(* Logix 5000 project; controller R5_CSS vendor 1 type 14 code 74 rev 19.11; software revision 19.01; part 17 of 20 *)
(* tags used below, declared in another part *)
   AlarmMaster : DINT;
   AllowHeatersWhenEmpty : BOOL;
   GTL_TDAHH_MinSP : REAL;
   HT_FAULT : BOOL;
   LC302 : LEVEL_CONTROL;   // COALESCER OIL CHAMBER LEVEL CONTROL
   MV301 : ValveControl_TwoWay;
   P302A : PUMP_CONTROL;
   P302B : PUMP_CONTROL;
   PID_JHE319 : PID;   // TEMPERATURE CONTROL OUPUT FOR JHE313B PID
   PID_JHE319_TON : TIMER;
   PID_TC215_TON : TIMER;
   PRU_TT404 : REAL[10];
   PRUA_READ : INT[30];
   TC112A : TEMP_CONTROL;
   TC121 : TEMP_CONTROL;
   TC121A : TEMP_CONTROL;   // GTL FROM PRUA TEMPERATURE CONTROL
   TC135 : TEMP_CONTROL;
   TC136 : TEMP_CONTROL;
   TC137 : TEMP_CONTROL;
   TC215 : TEMP_CONTROL;   // OVERHEAD CONDENSER CHILLED WATER TEMPERATURE TRANSMITTER CONTROL
   TC215_AUTO_ONS1 : BOOL;
   TC215_MANUAL_ONS1 : BOOL;
   TC313A : TEMP_CONTROL;   // PRIMARY COALESCER SEPARATOR TEMPERATURE CONTROL
   TC319 : TEMP_CONTROL;   // COALESCER OIL CHAMBER PROCESS TEMPERATURE CONTROL
   TC319_AUTO_Ons : BOOL;
   TC319_AUTO_Ons1 : BOOL;
   TC319_HeaterDisabled : BOOL;
   TC319_MANUAL_Ons : BOOL;
   TC319_START_TON : TIMER;
   TC319A : TEMP_CONTROL;   // COALESCER OIL CHAMBER SHEATH TEMPERATURE
   TCV215_PID : PID;
   TMR_FAULT : DINT;
(* MainProgram, continued *)

ROUTINE TC112A_CoalWaterHeaterBundleTemp   (* ladder *)
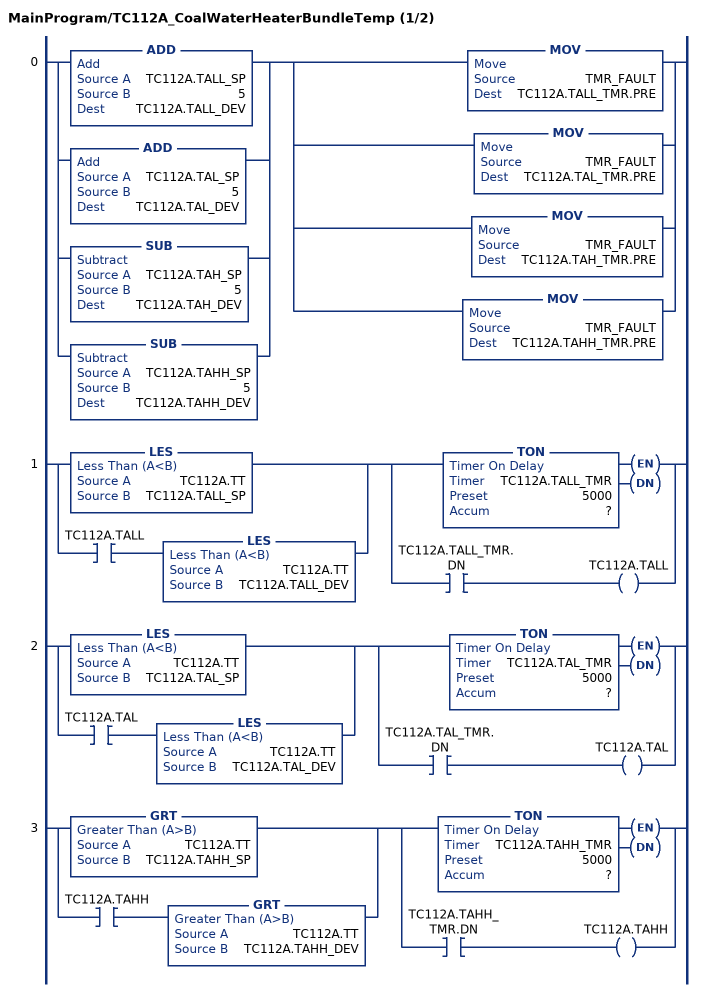
   0: [ADD(TC112A.TALL_SP,5,TC112A.TALL_DEV) ,ADD(TC112A.TAL_SP,5,TC112A.TAL_DEV) ,SUB(TC112A.TAH_SP,5,TC112A.TAH_DEV) ,SUB(TC112A.TAHH_SP,5,TC112A.TAHH_DEV) ][MOV(TMR_FAULT,TC112A.TALL_TMR.PRE) ,MOV(TMR_FAULT,TC112A.TAL_TMR.PRE) ,MOV(TMR_FAULT,TC112A.TAH_TMR.PRE) ,MOV(TMR_FAULT,TC112A.TAHH_TMR.PRE) ];
   1: [LES(TC112A.TT,TC112A.TALL_SP) ,XIC(TC112A.TALL) LES(TC112A.TT,TC112A.TALL_DEV) ][TON(TC112A.TALL_TMR,?,?) ,XIC(TC112A.TALL_TMR.DN) OTE(TC112A.TALL) ];
   2: [LES(TC112A.TT,TC112A.TAL_SP) ,XIC(TC112A.TAL) LES(TC112A.TT,TC112A.TAL_DEV) ][TON(TC112A.TAL_TMR,?,?) ,XIC(TC112A.TAL_TMR.DN) OTE(TC112A.TAL) ];
   3: [GRT(TC112A.TT,TC112A.TAHH_SP) ,XIC(TC112A.TAHH) GRT(TC112A.TT,TC112A.TAHH_DEV) ][TON(TC112A.TAHH_TMR,?,?) ,XIC(TC112A.TAHH_TMR.DN) OTE(TC112A.TAHH) ];
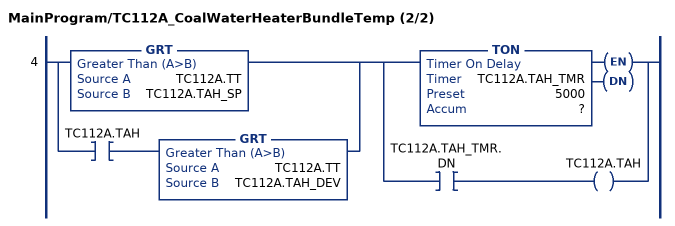
   4: [GRT(TC112A.TT,TC112A.TAH_SP) ,XIC(TC112A.TAH) GRT(TC112A.TT,TC112A.TAH_DEV) ][TON(TC112A.TAH_TMR,?,?) ,XIC(TC112A.TAH_TMR.DN) OTE(TC112A.TAH) ];
END_ROUTINE

ROUTINE TC135_GTL1_Temperature   (* ladder *)
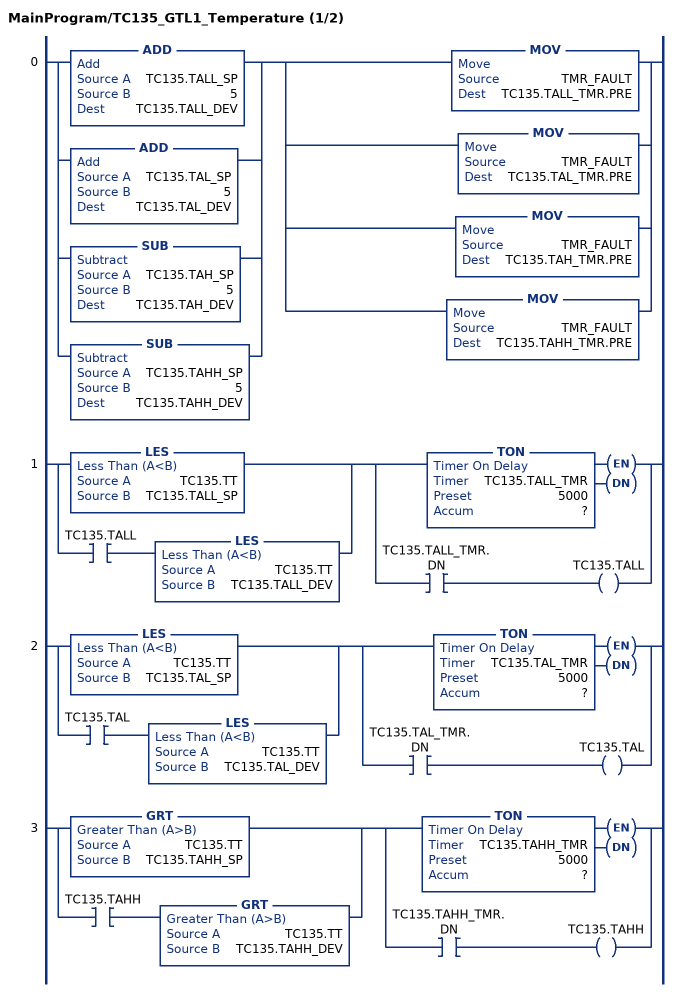
   0: [ADD(TC135.TALL_SP,5,TC135.TALL_DEV) ,ADD(TC135.TAL_SP,5,TC135.TAL_DEV) ,SUB(TC135.TAH_SP,5,TC135.TAH_DEV) ,SUB(TC135.TAHH_SP,5,TC135.TAHH_DEV) ][MOV(TMR_FAULT,TC135.TALL_TMR.PRE) ,MOV(TMR_FAULT,TC135.TAL_TMR.PRE) ,MOV(TMR_FAULT,TC135.TAH_TMR.PRE) ,MOV(TMR_FAULT,TC135.TAHH_TMR.PRE) ];
   1: [LES(TC135.TT,TC135.TALL_SP) ,XIC(TC135.TALL) LES(TC135.TT,TC135.TALL_DEV) ][TON(TC135.TALL_TMR,?,?) ,XIC(TC135.TALL_TMR.DN) OTE(TC135.TALL) ];
   2: [LES(TC135.TT,TC135.TAL_SP) ,XIC(TC135.TAL) LES(TC135.TT,TC135.TAL_DEV) ][TON(TC135.TAL_TMR,?,?) ,XIC(TC135.TAL_TMR.DN) OTE(TC135.TAL) ];
   3: [GRT(TC135.TT,TC135.TAHH_SP) ,XIC(TC135.TAHH) GRT(TC135.TT,TC135.TAHH_DEV) ][TON(TC135.TAHH_TMR,?,?) ,XIC(TC135.TAHH_TMR.DN) OTE(TC135.TAHH) ];
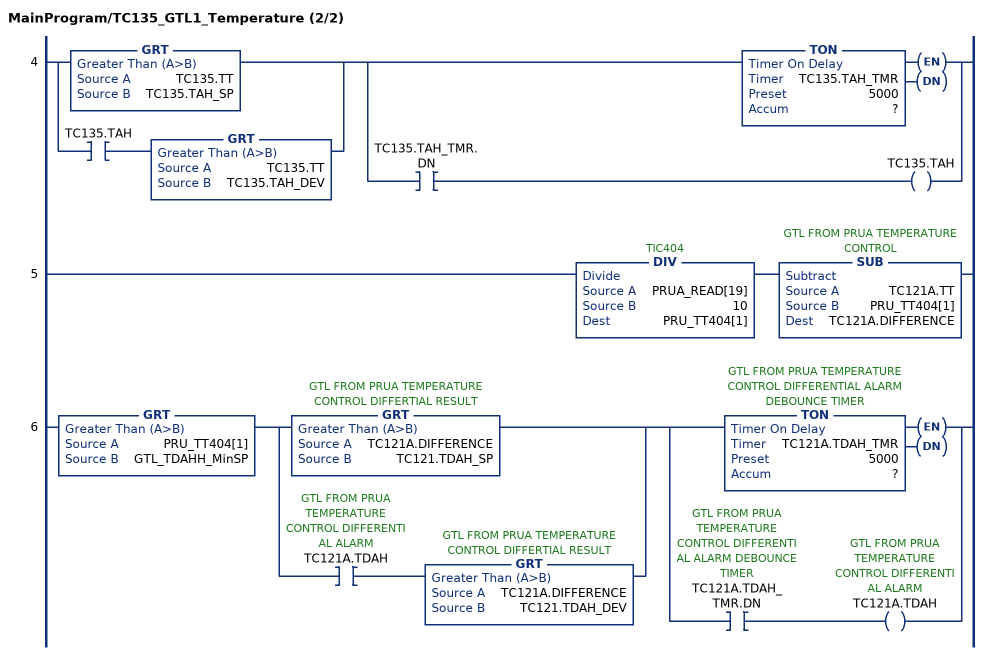
   4: [GRT(TC135.TT,TC135.TAH_SP) ,XIC(TC135.TAH) GRT(TC135.TT,TC135.TAH_DEV) ][TON(TC135.TAH_TMR,?,?) ,XIC(TC135.TAH_TMR.DN) OTE(TC135.TAH) ];
   5: DIV(PRUA_READ[19],10,PRU_TT404[1])SUB(TC121A.TT,PRU_TT404[1],TC121A.DIFFERENCE);
   6: GRT(PRU_TT404[1],GTL_TDAHH_MinSP)[GRT(TC121A.DIFFERENCE,TC121.TDAH_SP) ,XIC(TC121A.TDAH) GRT(TC121A.DIFFERENCE,TC121.TDAH_DEV) ][TON(TC121A.TDAH_TMR,?,?) ,XIC(TC121A.TDAH_TMR.DN) OTE(TC121A.TDAH) ];
END_ROUTINE

ROUTINE TC136_GTL2_Temperature   (* ladder *)
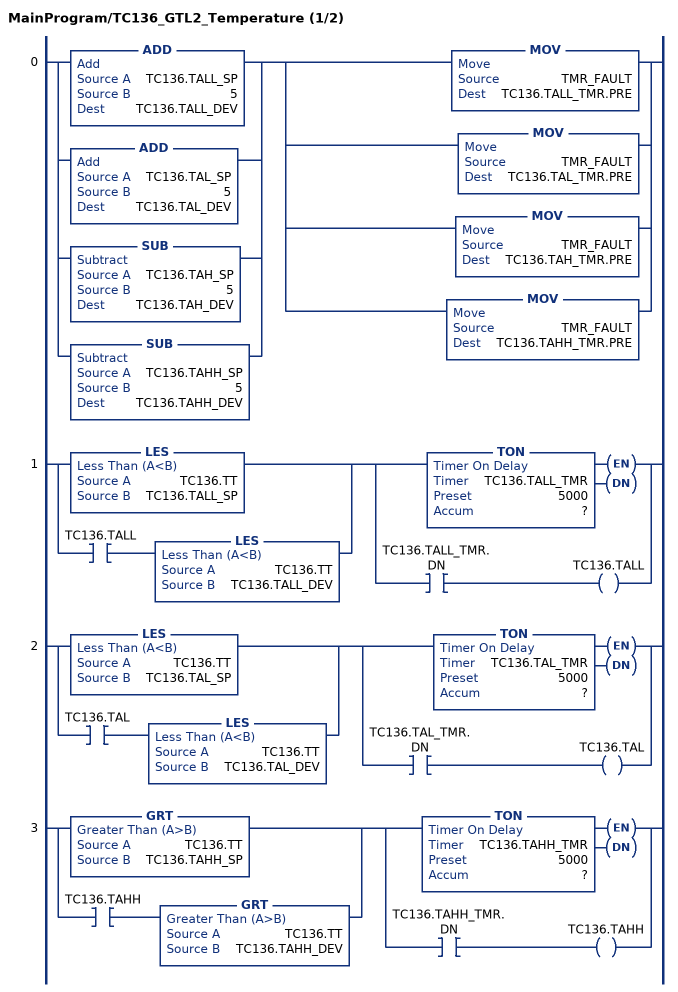
   0: [ADD(TC136.TALL_SP,5,TC136.TALL_DEV) ,ADD(TC136.TAL_SP,5,TC136.TAL_DEV) ,SUB(TC136.TAH_SP,5,TC136.TAH_DEV) ,SUB(TC136.TAHH_SP,5,TC136.TAHH_DEV) ][MOV(TMR_FAULT,TC136.TALL_TMR.PRE) ,MOV(TMR_FAULT,TC136.TAL_TMR.PRE) ,MOV(TMR_FAULT,TC136.TAH_TMR.PRE) ,MOV(TMR_FAULT,TC136.TAHH_TMR.PRE) ];
   1: [LES(TC136.TT,TC136.TALL_SP) ,XIC(TC136.TALL) LES(TC136.TT,TC136.TALL_DEV) ][TON(TC136.TALL_TMR,?,?) ,XIC(TC136.TALL_TMR.DN) OTE(TC136.TALL) ];
   2: [LES(TC136.TT,TC136.TAL_SP) ,XIC(TC136.TAL) LES(TC136.TT,TC136.TAL_DEV) ][TON(TC136.TAL_TMR,?,?) ,XIC(TC136.TAL_TMR.DN) OTE(TC136.TAL) ];
   3: [GRT(TC136.TT,TC136.TAHH_SP) ,XIC(TC136.TAHH) GRT(TC136.TT,TC136.TAHH_DEV) ][TON(TC136.TAHH_TMR,?,?) ,XIC(TC136.TAHH_TMR.DN) OTE(TC136.TAHH) ];
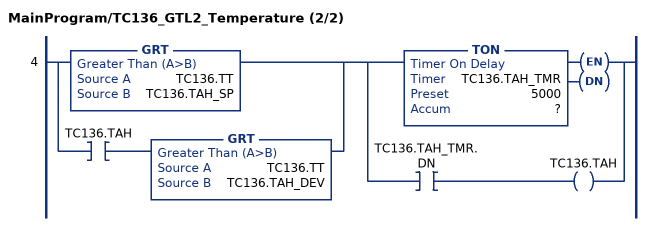
   4: [GRT(TC136.TT,TC136.TAH_SP) ,XIC(TC136.TAH) GRT(TC136.TT,TC136.TAH_DEV) ][TON(TC136.TAH_TMR,?,?) ,XIC(TC136.TAH_TMR.DN) OTE(TC136.TAH) ];
END_ROUTINE

ROUTINE TC137_GTL3_Temperature   (* ladder *)
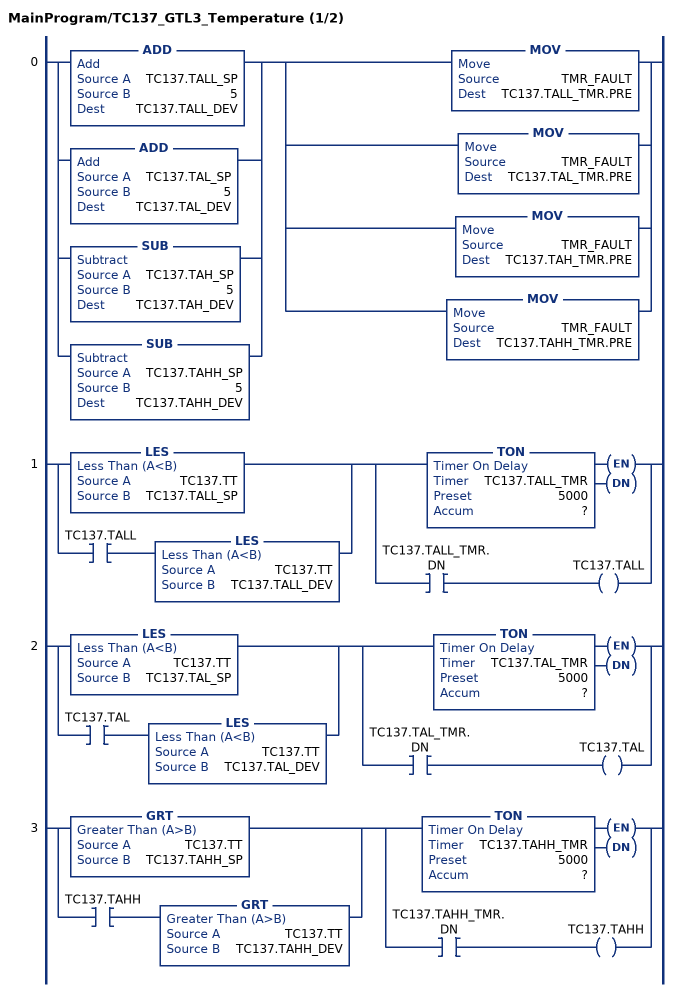
   0: [ADD(TC137.TALL_SP,5,TC137.TALL_DEV) ,ADD(TC137.TAL_SP,5,TC137.TAL_DEV) ,SUB(TC137.TAH_SP,5,TC137.TAH_DEV) ,SUB(TC137.TAHH_SP,5,TC137.TAHH_DEV) ][MOV(TMR_FAULT,TC137.TALL_TMR.PRE) ,MOV(TMR_FAULT,TC137.TAL_TMR.PRE) ,MOV(TMR_FAULT,TC137.TAH_TMR.PRE) ,MOV(TMR_FAULT,TC137.TAHH_TMR.PRE) ];
   1: [LES(TC137.TT,TC137.TALL_SP) ,XIC(TC137.TALL) LES(TC137.TT,TC137.TALL_DEV) ][TON(TC137.TALL_TMR,?,?) ,XIC(TC137.TALL_TMR.DN) OTE(TC137.TALL) ];
   2: [LES(TC137.TT,TC137.TAL_SP) ,XIC(TC137.TAL) LES(TC137.TT,TC137.TAL_DEV) ][TON(TC137.TAL_TMR,?,?) ,XIC(TC137.TAL_TMR.DN) OTE(TC137.TAL) ];
   3: [GRT(TC137.TT,TC137.TAHH_SP) ,XIC(TC137.TAHH) GRT(TC137.TT,TC137.TAHH_DEV) ][TON(TC137.TAHH_TMR,?,?) ,XIC(TC137.TAHH_TMR.DN) OTE(TC137.TAHH) ];
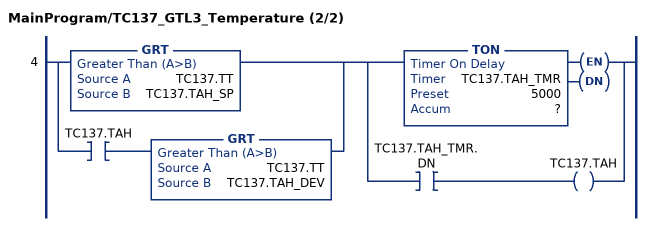
   4: [GRT(TC137.TT,TC137.TAH_SP) ,XIC(TC137.TAH) GRT(TC137.TT,TC137.TAH_DEV) ][TON(TC137.TAH_TMR,?,?) ,XIC(TC137.TAH_TMR.DN) OTE(TC137.TAH) ];
END_ROUTINE

ROUTINE TC215_OverheadCondTemp_PID   (* ladder *)
// NonCondensable Process Gas Temperature Control
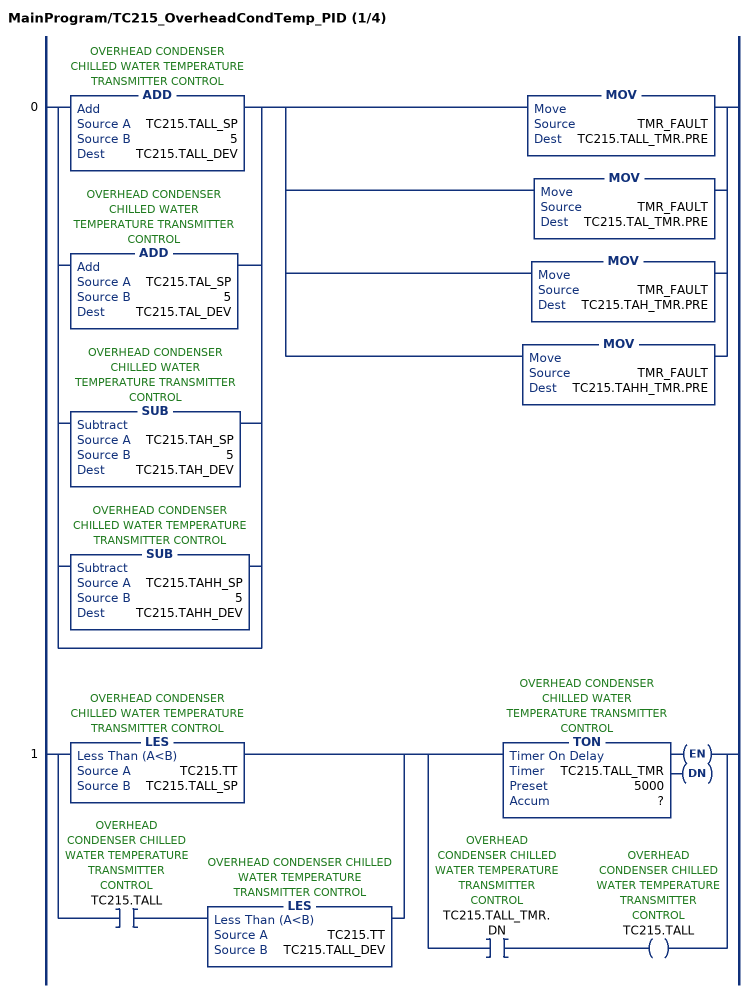
   0: [ADD(TC215.TALL_SP,5,TC215.TALL_DEV) ,ADD(TC215.TAL_SP,5,TC215.TAL_DEV) ,SUB(TC215.TAH_SP,5,TC215.TAH_DEV) ,SUB(TC215.TAHH_SP,5,TC215.TAHH_DEV) ,][MOV(TMR_FAULT,TC215.TALL_TMR.PRE) ,MOV(TMR_FAULT,TC215.TAL_TMR.PRE) ,MOV(TMR_FAULT,TC215.TAH_TMR.PRE) ,MOV(TMR_FAULT,TC215.TAHH_TMR.PRE) ];
   1: [LES(TC215.TT,TC215.TALL_SP) ,XIC(TC215.TALL) LES(TC215.TT,TC215.TALL_DEV) ][TON(TC215.TALL_TMR,?,?) ,XIC(TC215.TALL_TMR.DN) OTE(TC215.TALL) ];
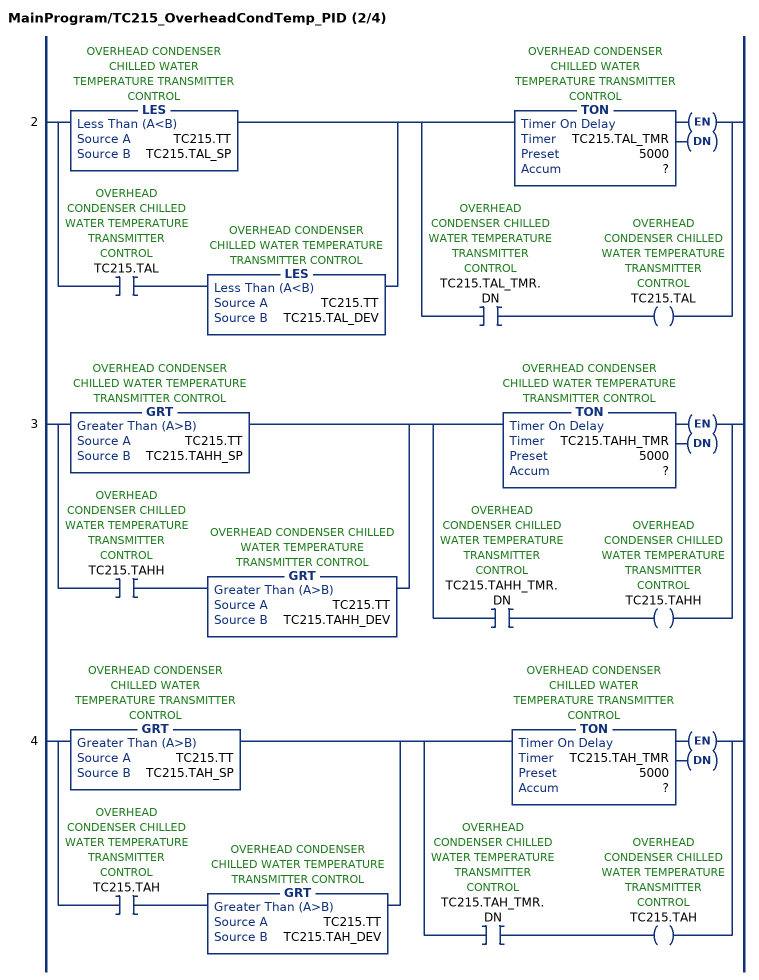
   2: [LES(TC215.TT,TC215.TAL_SP) ,XIC(TC215.TAL) LES(TC215.TT,TC215.TAL_DEV) ][TON(TC215.TAL_TMR,?,?) ,XIC(TC215.TAL_TMR.DN) OTE(TC215.TAL) ];
   3: [GRT(TC215.TT,TC215.TAHH_SP) ,XIC(TC215.TAHH) GRT(TC215.TT,TC215.TAHH_DEV) ][TON(TC215.TAHH_TMR,?,?) ,XIC(TC215.TAHH_TMR.DN) OTE(TC215.TAHH) ];
   4: [GRT(TC215.TT,TC215.TAH_SP) ,XIC(TC215.TAH) GRT(TC215.TT,TC215.TAH_DEV) ][TON(TC215.TAH_TMR,?,?) ,XIC(TC215.TAH_TMR.DN) OTE(TC215.TAH) ];
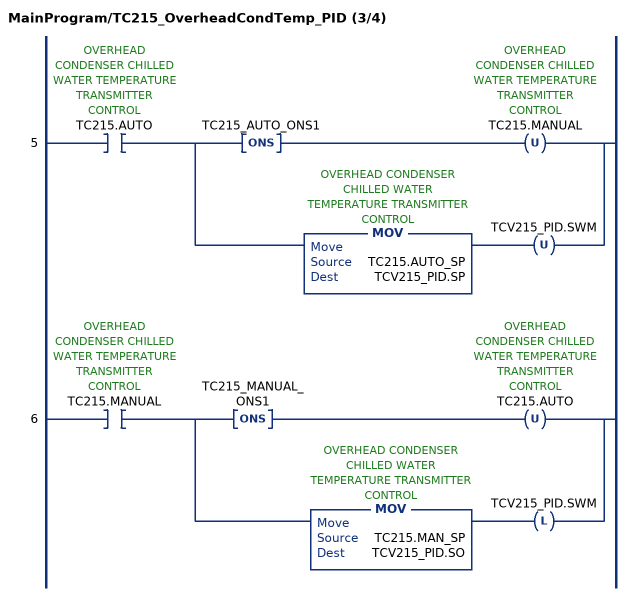
   5: XIC(TC215.AUTO)[ONS(TC215_AUTO_ONS1) OTU(TC215.MANUAL) ,MOV(TC215.AUTO_SP,TCV215_PID.SP) OTU(TCV215_PID.SWM) ];
   6: XIC(TC215.MANUAL)[ONS(TC215_MANUAL_ONS1) OTU(TC215.AUTO) ,MOV(TC215.MAN_SP,TCV215_PID.SO) OTL(TCV215_PID.SWM) ];
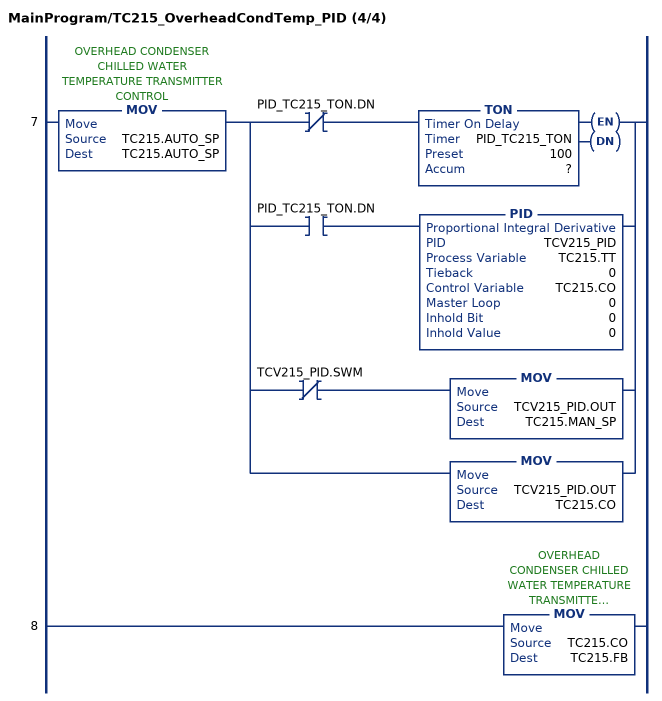
   7: MOV(TC215.AUTO_SP,TC215.AUTO_SP)[XIO(PID_TC215_TON.DN) TON(PID_TC215_TON,?,?) ,XIC(PID_TC215_TON.DN) PID(TCV215_PID,TC215.TT,0,TC215.CO,0,0,0) ,XIO(TCV215_PID.SWM) MOV(TCV215_PID.OUT,TC215.MAN_SP) ,MOV(TCV215_PID.OUT,TC215.CO) ];
   8: MOV(TC215.CO,TC215.FB);
END_ROUTINE

ROUTINE TC313A_CoalPriChamberTemperature   (* ladder *)
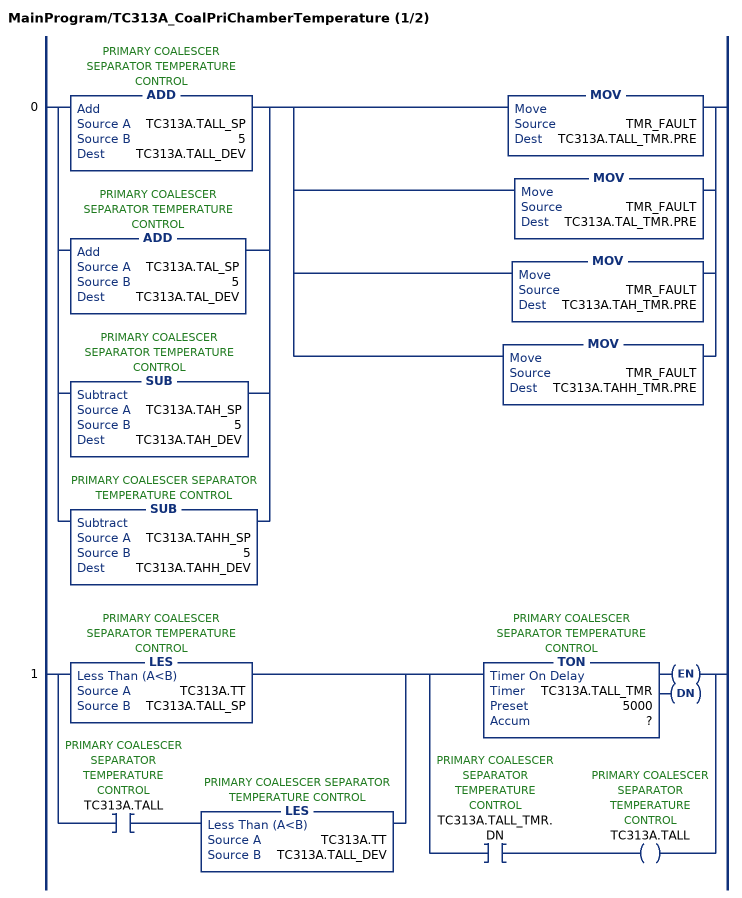
   0: [ADD(TC313A.TALL_SP,5,TC313A.TALL_DEV) ,ADD(TC313A.TAL_SP,5,TC313A.TAL_DEV) ,SUB(TC313A.TAH_SP,5,TC313A.TAH_DEV) ,SUB(TC313A.TAHH_SP,5,TC313A.TAHH_DEV) ][MOV(TMR_FAULT,TC313A.TALL_TMR.PRE) ,MOV(TMR_FAULT,TC313A.TAL_TMR.PRE) ,MOV(TMR_FAULT,TC313A.TAH_TMR.PRE) ,MOV(TMR_FAULT,TC313A.TAHH_TMR.PRE) ];
   1: [LES(TC313A.TT,TC313A.TALL_SP) ,XIC(TC313A.TALL) LES(TC313A.TT,TC313A.TALL_DEV) ][TON(TC313A.TALL_TMR,?,?) ,XIC(TC313A.TALL_TMR.DN) OTE(TC313A.TALL) ];
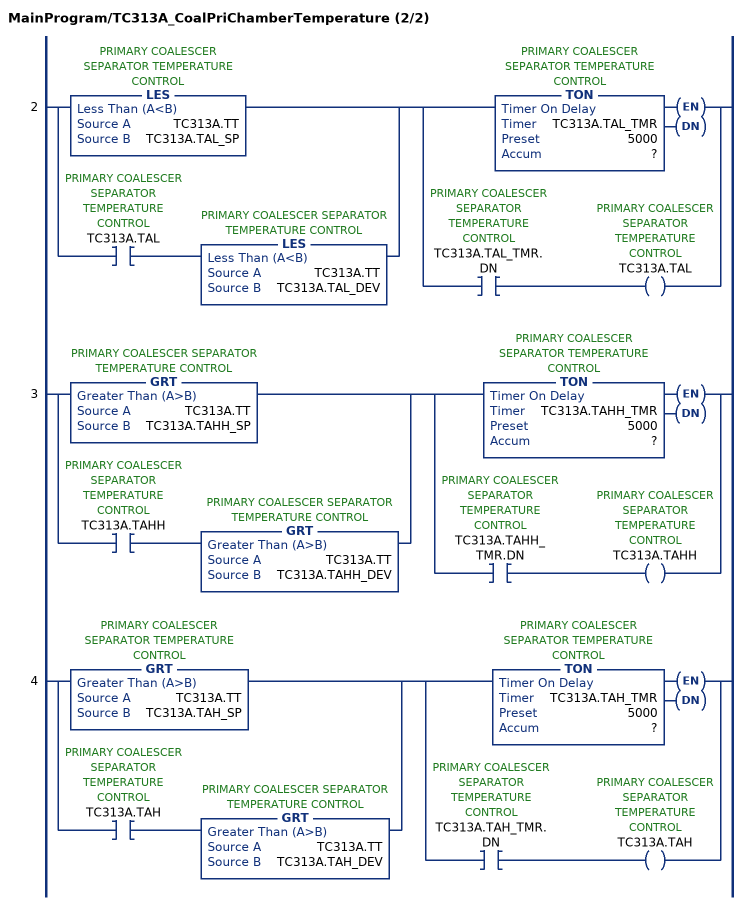
   2: [LES(TC313A.TT,TC313A.TAL_SP) ,XIC(TC313A.TAL) LES(TC313A.TT,TC313A.TAL_DEV) ][TON(TC313A.TAL_TMR,?,?) ,XIC(TC313A.TAL_TMR.DN) OTE(TC313A.TAL) ];
   3: [GRT(TC313A.TT,TC313A.TAHH_SP) ,XIC(TC313A.TAHH) GRT(TC313A.TT,TC313A.TAHH_DEV) ][TON(TC313A.TAHH_TMR,?,?) ,XIC(TC313A.TAHH_TMR.DN) OTE(TC313A.TAHH) ];
   4: [GRT(TC313A.TT,TC313A.TAH_SP) ,XIC(TC313A.TAH) GRT(TC313A.TT,TC313A.TAH_DEV) ][TON(TC313A.TAH_TMR,?,?) ,XIC(TC313A.TAH_TMR.DN) OTE(TC313A.TAH) ];
END_ROUTINE

ROUTINE TC319_OilProductTemperature_PID   (* ladder *)
// OIL TRANSFER CHAMBER HEAT CONTROL
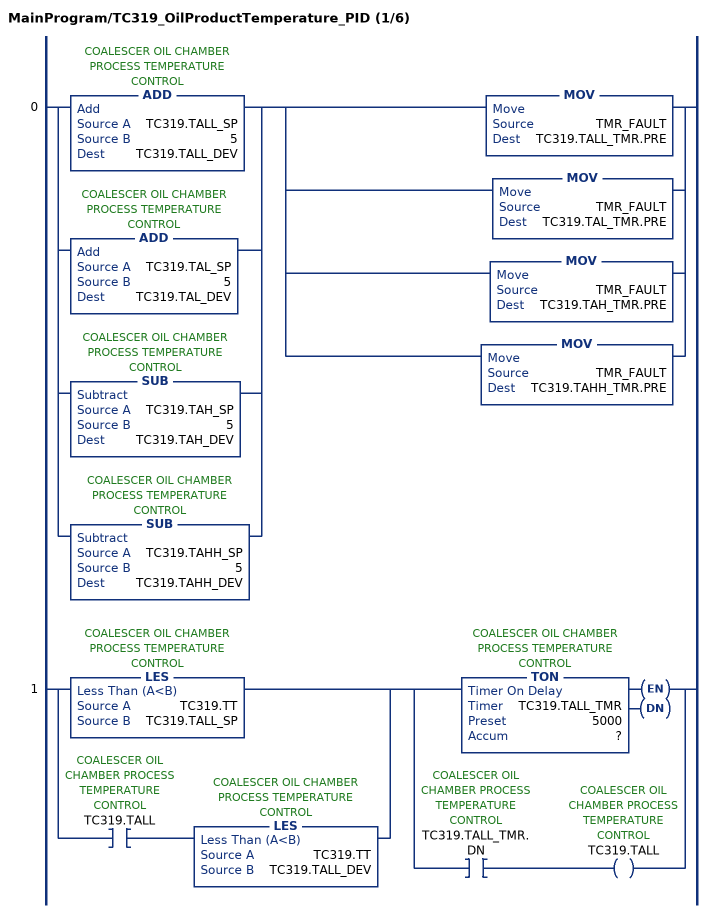
   0: [ADD(TC319.TALL_SP,5,TC319.TALL_DEV) ,ADD(TC319.TAL_SP,5,TC319.TAL_DEV) ,SUB(TC319.TAH_SP,5,TC319.TAH_DEV) ,SUB(TC319.TAHH_SP,5,TC319.TAHH_DEV) ][MOV(TMR_FAULT,TC319.TALL_TMR.PRE) ,MOV(TMR_FAULT,TC319.TAL_TMR.PRE) ,MOV(TMR_FAULT,TC319.TAH_TMR.PRE) ,MOV(TMR_FAULT,TC319.TAHH_TMR.PRE) ];
   1: [LES(TC319.TT,TC319.TALL_SP) ,XIC(TC319.TALL) LES(TC319.TT,TC319.TALL_DEV) ][TON(TC319.TALL_TMR,?,?) ,XIC(TC319.TALL_TMR.DN) OTE(TC319.TALL) ];
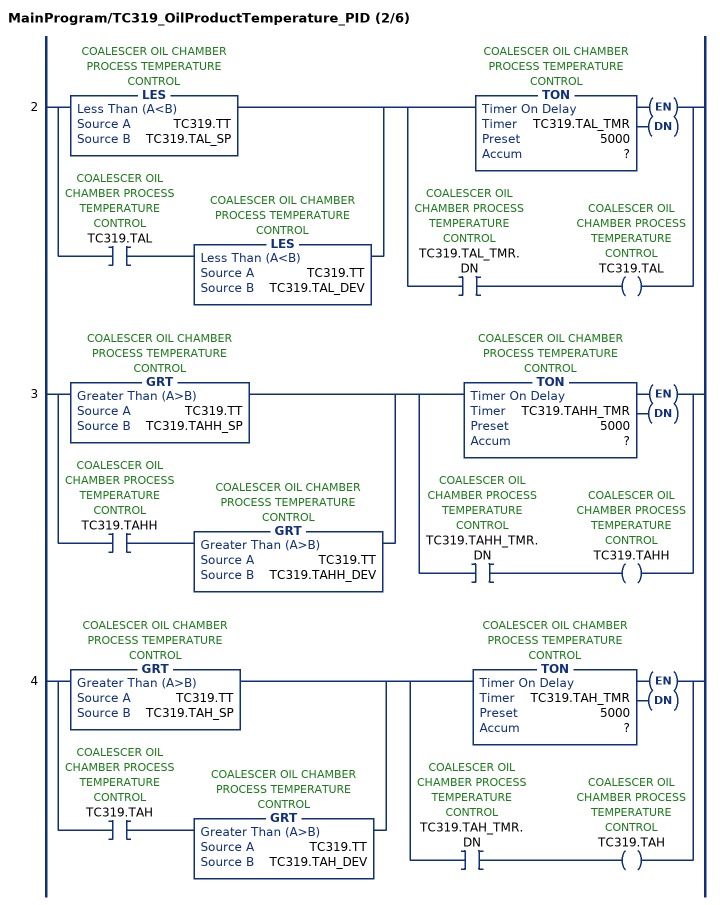
   2: [LES(TC319.TT,TC319.TAL_SP) ,XIC(TC319.TAL) LES(TC319.TT,TC319.TAL_DEV) ][TON(TC319.TAL_TMR,?,?) ,XIC(TC319.TAL_TMR.DN) OTE(TC319.TAL) ];
   3: [GRT(TC319.TT,TC319.TAHH_SP) ,XIC(TC319.TAHH) GRT(TC319.TT,TC319.TAHH_DEV) ][TON(TC319.TAHH_TMR,?,?) ,XIC(TC319.TAHH_TMR.DN) OTE(TC319.TAHH) ];
   4: [GRT(TC319.TT,TC319.TAH_SP) ,XIC(TC319.TAH) GRT(TC319.TT,TC319.TAH_DEV) ][TON(TC319.TAH_TMR,?,?) ,XIC(TC319.TAH_TMR.DN) OTE(TC319.TAH) ];
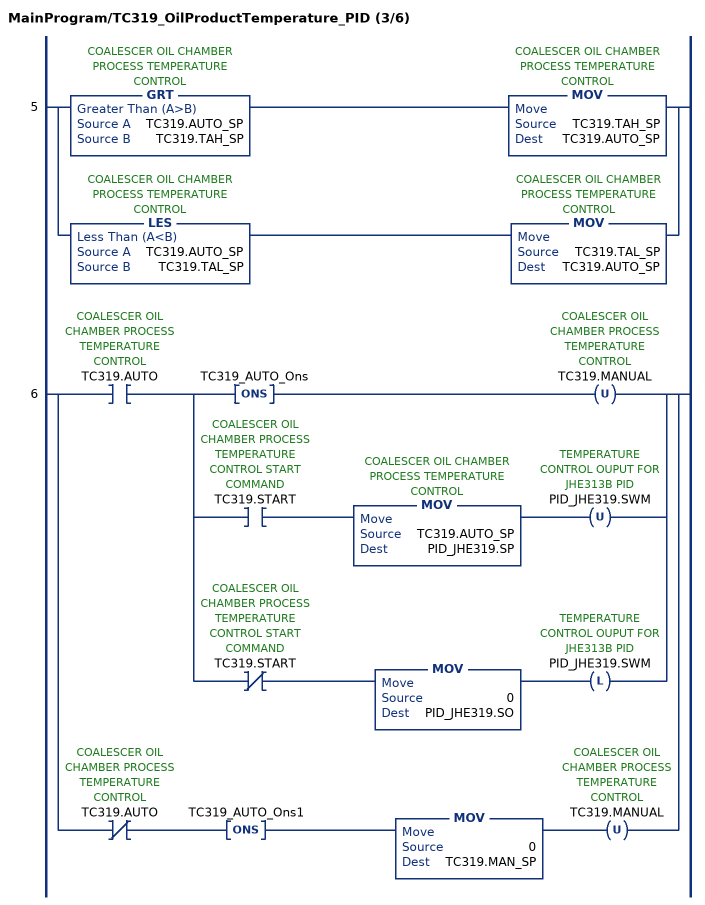
   5: [GRT(TC319.AUTO_SP,TC319.TAH_SP) MOV(TC319.TAH_SP,TC319.AUTO_SP) ,LES(TC319.AUTO_SP,TC319.TAL_SP) MOV(TC319.TAL_SP,TC319.AUTO_SP) ];
   6: [XIC(TC319.AUTO) [ONS(TC319_AUTO_Ons) OTU(TC319.MANUAL) ,XIC(TC319.START) MOV(TC319.AUTO_SP,PID_JHE319.SP) OTU(PID_JHE319.SWM) ,XIO(TC319.START) MOV(0,PID_JHE319.SO) OTL(PID_JHE319.SWM) ] ,XIO(TC319.AUTO) ONS(TC319_AUTO_Ons1) MOV(0,TC319.MAN_SP) OTU(TC319.MANUAL) ];
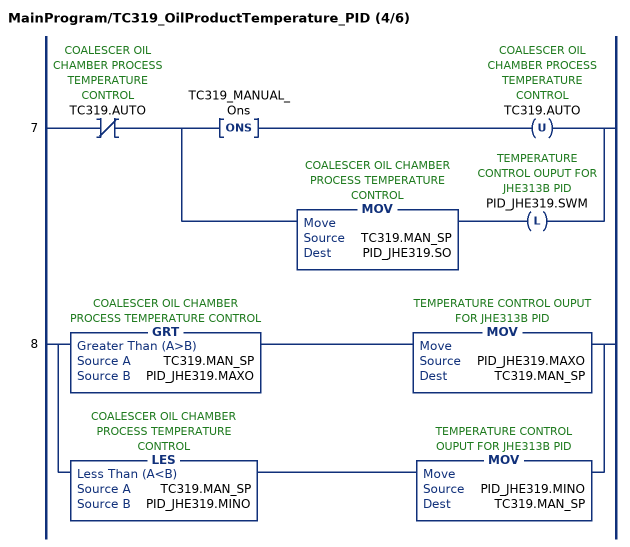
   7: XIO(TC319.AUTO)[ONS(TC319_MANUAL_Ons) OTU(TC319.AUTO) ,MOV(TC319.MAN_SP,PID_JHE319.SO) OTL(PID_JHE319.SWM) ];
   8: [GRT(TC319.MAN_SP,PID_JHE319.MAXO) MOV(PID_JHE319.MAXO,TC319.MAN_SP) ,LES(TC319.MAN_SP,PID_JHE319.MINO) MOV(PID_JHE319.MINO,TC319.MAN_SP) ];
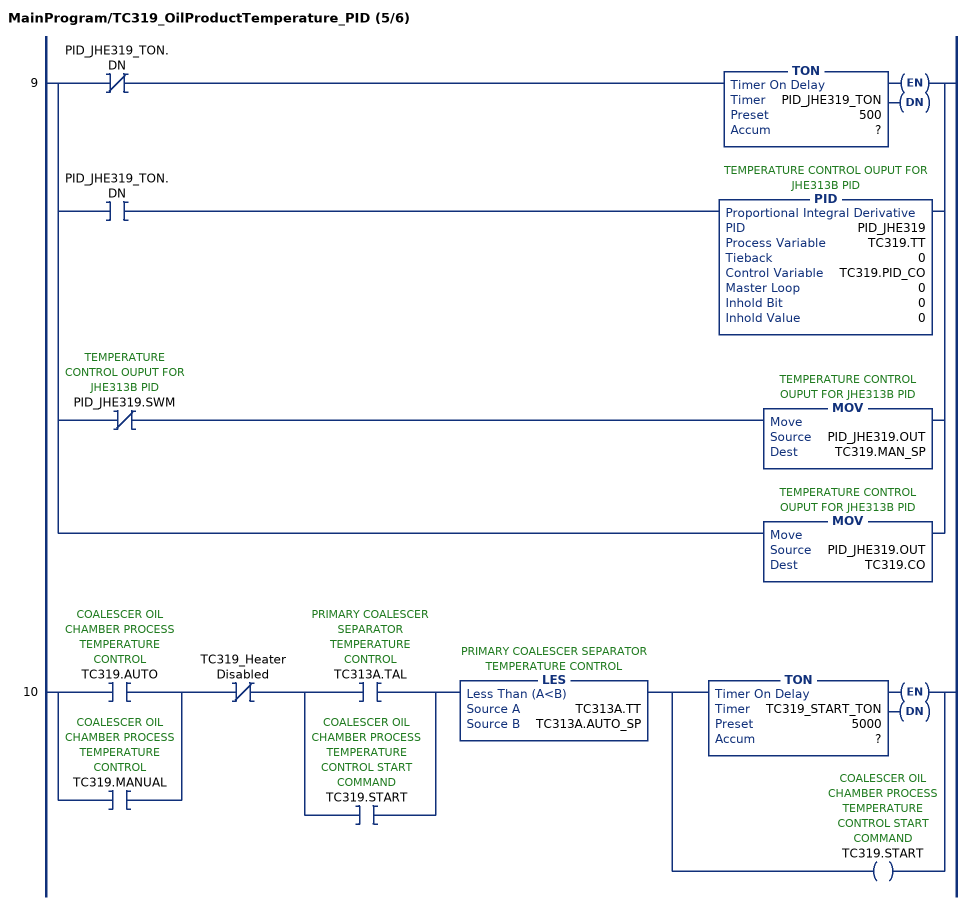
   9: [XIO(PID_JHE319_TON.DN) TON(PID_JHE319_TON,?,?) ,XIC(PID_JHE319_TON.DN) PID(PID_JHE319,TC319.TT,0,TC319.PID_CO,0,0,0) ,XIO(PID_JHE319.SWM) MOV(PID_JHE319.OUT,TC319.MAN_SP) ,MOV(PID_JHE319.OUT,TC319.CO) ];
   10: [XIC(TC319.AUTO) ,XIC(TC319.MANUAL) ]XIO(TC319_HeaterDisabled)[XIC(TC313A.TAL) ,XIC(TC319.START) ]LES(TC313A.TT,TC313A.AUTO_SP)[TON(TC319_START_TON,?,?) ,OTE(TC319.START) ];
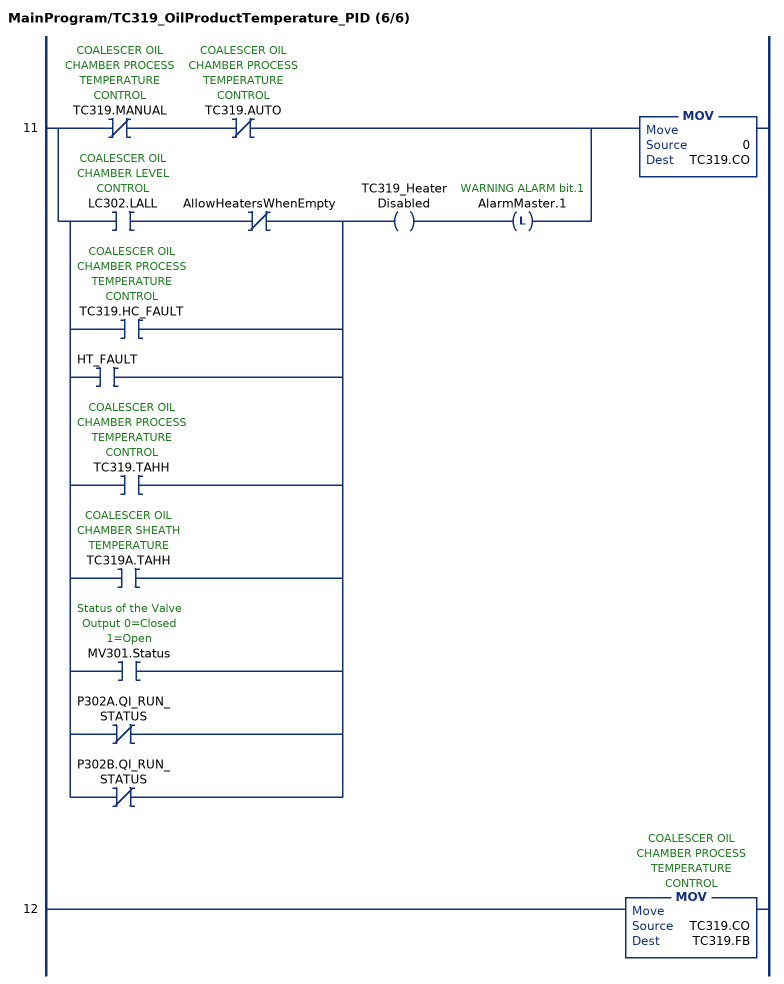
   11: [XIO(TC319.MANUAL) XIO(TC319.AUTO) ,[XIC(LC302.LALL) XIO(AllowHeatersWhenEmpty) ,XIC(TC319.HC_FAULT) ,XIC(HT_FAULT) ,XIC(TC319.TAHH) ,XIC(TC319A.TAHH) ,XIC(MV301.Status) ,XIO(P302A.QI_RUN_STATUS) ,XIO(P302B.QI_RUN_STATUS) ] OTE(TC319_HeaterDisabled) OTL(AlarmMaster.1) ]MOV(0,TC319.CO);
   12: MOV(TC319.CO,TC319.FB);
END_ROUTINE
